# EPICS substitutions: ek9000App/Db/EL3174.substitutions
file EL3174.template
{       pattern
        {
                TERMINAL,

        }
        {
        }
}
